TYPE st_TeltonikaEvents :
STRUCT
	b_MBCommWarning		:	BOOL;
	b_MBCommError		:	BOOL;
	b_NoSimWarning		:	BOOL;
	b_NoNetworkWarning	: 	BOOL;
	b_noGPSFixWarning	:	BOOL;
	b_SMSNotSendError	:	BOOL; 
	b_NoSMSNumberAvailable	:	BOOL;
END_STRUCT
END_TYPE

(* stored: Version 1.1.0.1, ProductVersion 3.1.4024.12
   DUT st_TeltonikaEvents: Id {cd092dc8-29f2-4e3d-a6b8-43e406070d5a} *)
